TYPE ST_RinseChannel :
STRUCT
	nPumpNr	 	: USINT;
	nValveNr	: USINT;
	nStartSpeed	: USINT;
	nRatedSpeed : USINT;
	nStartTime	: UINT;
END_STRUCT
END_TYPE

(* stored: Version 1.1.0.1, ProductVersion 3.1.4020.6
   DUT ST_RinseChannel: Id {a72cf7d4-5ee0-4bb5-bfa8-667d2c02c963} *)
